// Mitsubishi GX Works2 project: wind   PLC: FX3U/FX3UC

PROGRAM MAIN
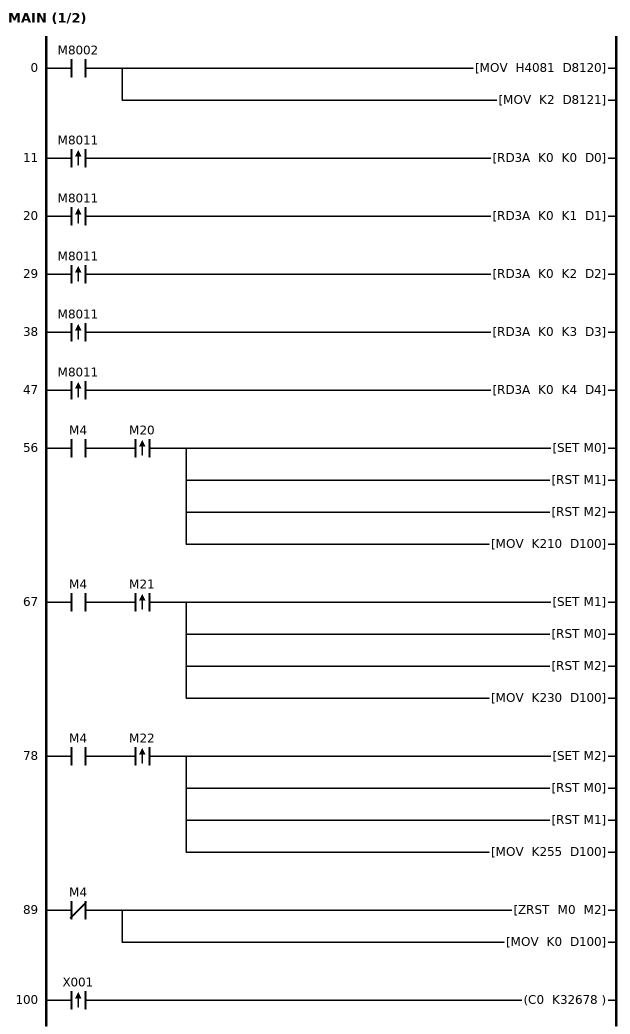
0     LD      M8002
      MOV     H4081 D8120
      MOV     K2 D8121
11    LDP     M8011
      RD3A    K0 K0 D0
20    LDP     M8011
      RD3A    K0 K1 D1
29    LDP     M8011
      RD3A    K0 K2 D2
38    LDP     M8011
      RD3A    K0 K3 D3
47    LDP     M8011
      RD3A    K0 K4 D4
56    LD      M4
      ANDP    M20
      SET     M0
      RST     M1
      RST     M2
      MOV     K210 D100
67    LD      M4
      ANDP    M21
      SET     M1
      RST     M0
      RST     M2
      MOV     K230 D100
78    LD      M4
      ANDP    M22
      SET     M2
      RST     M0
      RST     M1
      MOV     K255 D100
89    LDI     M4
      ZRST    M0 M2
      MOV     K0 D100
100   LDP     X001
      OUT     C0 K32678
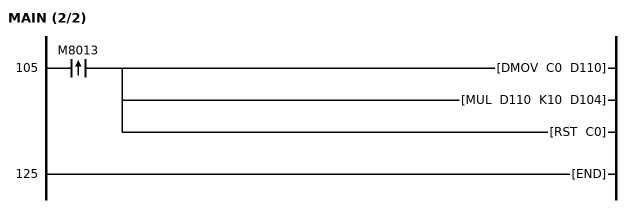
105   LDP     M8013
      DMOV    C0 D110
      MUL     D110 K10 D104
      RST     C0
125   END
END_PROGRAM
